TYPE INT_INDEX : INT(0..32767); END_TYPE

(* stored: Version 1.1.0.1
   DUT INT_INDEX: Id {32988081-e0ea-477c-b49b-40f4213cf20d} *)
